FUNCTION_BLOCK fBDISCRETE_PID
VAR_INPUT
	Setpoint:REAL;         // SetPoint
    Kp:REAL;               // Kp  Proportional gain
	Ki:REAL;               // Ki  Integrated gain
	Kd:REAL;               // Kd  Derivative gain
	Nfilter       : REAL;  // Lowpass Filter Coeff 
	Yprocess      : REAL;  // Process Output
	Auto_Mode     : BOOL;  // PId enable if true (closed loop )
	MV_max_sat    : REAL;  // Maximum Saturation
	MV_min_sat    : REAL;  // Minimum Saturation
	xExt_Error    : BOOL;  // External error 
	
END_VAR
VAR_OUTPUT
	MV_out        : REAL;    // Controller output
	Inposition    : BOOL;    //  2% Settled. not implemented yet. 
END_VAR
VAR
	T1     : REAL :=0;
	Perr, Perr1, Perr2 : REAL ;
    A,B,C  :REAL;
	MV_out1:REAL;
	Tsample:REAL := 0.01;
END_VAR

//
IF T1 = 0 THEN
	MV_out:=0;     // no bias offset controller
END_IF

T1:=Tsample; 
Perr:= Setpoint - Yprocess; // Current error e[k]
//
// Constant Coefficients including the Parameters Kp , Ki, Kd and Tsample
//        Your PID Controller algorithm starts here
//
// A:= (Kp +Ki*(Tsample/2)+(Kd/Tsample));
// B:= (-Kp +Ki*(Tsample/2)-(2*Kd/Tsample));
// C:=  Kd/Tsample;
//
//   Mv_out:= MV_out1 + A*perr +B*perr1 + C*perr2:                                // PID Controller
//
MV_out:=  Kp * Perr;  // P-Controller 

// Update  samples 
MV_out1:= MV_out;      // MV_out[k-1] 
Perr2  := Perr1;       // e[k-2]
Perr1  := Perr;        // e[k-1]

//  PID  is not Enabled 
IF NOT Auto_Mode THEN
	MV_Out:= Setpoint;   ///  Open loop 
END_IF

//    PID  output saturation 
IF Mv_out < MV_min_sat THEN
	Mv_out:= MV_min_sat;
END_IF
IF Mv_out >  MV_max_sat THEN
	Mv_out:= MV_max_sat;
END_IF

END_FUNCTION_BLOCK

(* stored: Version 1.1.0.1, ProductVersion 3.1.4024.2
   POU fBDISCRETE_PID: Id {6d63eba5-46e9-49ad-b783-0b876d499556}, SpecialFunc None *)
